// TIA Portal V19 export
FUNCTION_BLOCK "System_FB"   // FB3, LAD
TITLE = System bits
AUTHOR : Piemme
FAMILY : System
VERSION : 1.2
// stored: Access Published, MemoryReserve 100, SetENOAutomatically false
   VAR_INPUT
      PbLampTest : Bool;
   END_VAR
   VAR
      Ton0 : IEC_TIMER;
      wFrequencyGen : Word;
      wFrequencyLampTest : Word;
      PreviuosCycleTime : "CpuPreviuosCycleTime";
   END_VAR
   VAR_TEMP   // added for the SCL form of the ladder/FBD networks
      _w1 : Bool;
   END_VAR
BEGIN

REGION Network 1 (SCL): Info
   //=============================================================================
   //PM FORMING
   //-----------------------------------------------------------------------------
   // Library: StandardBlocks
   // Tested with: S7-1518TF
   // Engineering: TIA Portal V18
   // Restrictions: -
   // Requirements: S7-1500
   // Functionality: System management
   //
   // v1.0.0  28/12/2022 
   //=============================================================================
END_REGION

REGION Network 2: Set/Rst bits always true / false
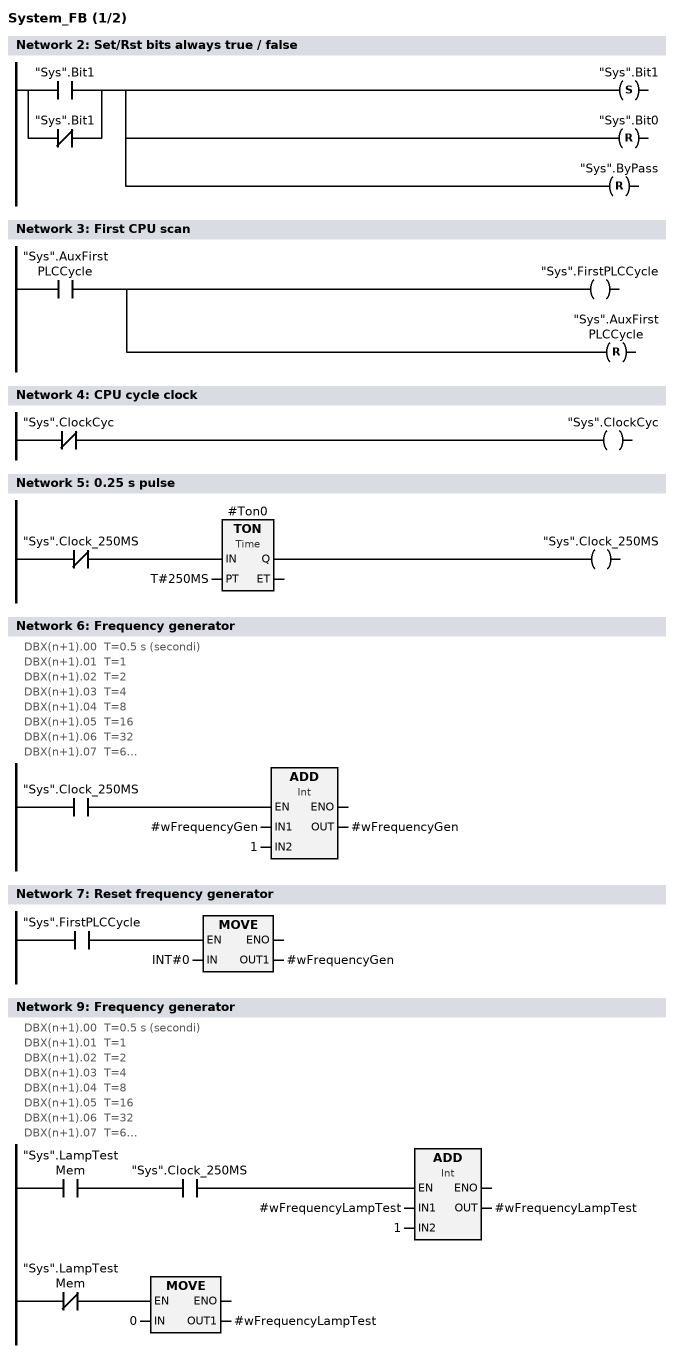
   RUNG wire#powerrail
      Contact( "Sys".Bit1 )
      wire#w1
      S_Coil( "Sys".Bit1 )
   END_RUNG
   RUNG wire#powerrail
      I_Contact( "Sys".Bit1 )
   END_RUNG wire#w1
   RUNG wire#w1
      R_Coil( "Sys".Bit0 )
   END_RUNG
   RUNG wire#w1
      R_Coil( "Sys".ByPass )
   END_RUNG
   // the same network as SCL:
   #_w1 := "Sys".Bit1 OR NOT "Sys".Bit1;
   IF #_w1 THEN
       "Sys".Bit1 := TRUE;
       "Sys".Bit0 := FALSE;
       "Sys".ByPass := FALSE;
   END_IF;
END_REGION

REGION Network 3: First CPU scan
   RUNG wire#powerrail
      Contact( "Sys".AuxFirstPLCCycle )
      wire#w1
      Coil( "Sys".FirstPLCCycle )
   END_RUNG
   RUNG wire#w1
      R_Coil( "Sys".AuxFirstPLCCycle )
   END_RUNG
   // the same network as SCL:
   "Sys".FirstPLCCycle := "Sys".AuxFirstPLCCycle;
   IF "Sys".AuxFirstPLCCycle THEN "Sys".AuxFirstPLCCycle := FALSE; END_IF;
END_REGION

REGION Network 4: CPU cycle clock
   RUNG wire#powerrail
      I_Contact( "Sys".ClockCyc )
      Coil( "Sys".ClockCyc )
   END_RUNG
   // the same network as SCL:
   "Sys".ClockCyc := NOT "Sys".ClockCyc;
END_REGION

REGION Network 5: 0.25 s pulse
   RUNG wire#powerrail
      I_Contact( "Sys".Clock_250MS )
      { S7_Templates := "time_type := Time" } #Ton0.TON(pt := T#250MS, et =>)
      Coil( "Sys".Clock_250MS )
   END_RUNG
   // the same network as SCL:
   #Ton0.TON(IN := NOT "Sys".Clock_250MS, PT := T#250MS);
   "Sys".Clock_250MS := #Ton0.Q;
END_REGION

REGION Network 6: Frequency generator
   // DBX(n+1).00  T=0.5 s (secondi)
   // DBX(n+1).01  T=1
   // DBX(n+1).02  T=2
   // DBX(n+1).03  T=4
   // DBX(n+1).04  T=8
   // DBX(n+1).05  T=16
   // DBX(n+1).06  T=32
   // DBX(n+1).07  T=64     
   // DBX  (n).00  T=128    (2 M)
   // DBX  (n).01  T=256    (4.2 M)
   // DBX  (n).02  T=512    (8.5 M)
   // DBX  (n).03  T=1024   (17 M)
   // DBX  (n).04  T=2048   (34.1 M)
   // DBX  (n).05  T=4096   (68.2 M)
   // DBX  (n).06  T=8192   (2 H)
   // DBX  (n).07  T=16384  (4 H)
   RUNG wire#powerrail
      Contact( "Sys".Clock_250MS )
      { S7_Templates := "SrcType := Int"; S7_GenerateENO := "TRUE" } Add(in1 := #wFrequencyGen, in2 := 1, out => #wFrequencyGen)
   END_RUNG
   // the same network as SCL:
   IF "Sys".Clock_250MS THEN #wFrequencyGen := #wFrequencyGen + 1; END_IF;
END_REGION

REGION Network 7: Reset frequency generator
   RUNG wire#powerrail
      Contact( "Sys".FirstPLCCycle )
      { S7_GenerateENO := "TRUE" } Move(in := INT#0, out1 => #wFrequencyGen)
   END_RUNG
   // the same network as SCL:
   IF "Sys".FirstPLCCycle THEN #wFrequencyGen := INT#0; END_IF;
END_REGION

REGION Network 8 (SCL): MB of clocks / Clocks
   "Sys".Clock_500MS := #wFrequencyGen.%X0;
   "Sys".Clock_1S := #wFrequencyGen.%X1;
   "Sys".Clock_2S := #wFrequencyGen.%X2;
   "Sys".Clock_4S := #wFrequencyGen.%X3;
   "Sys".Clock_8S := #wFrequencyGen.%X4;
   "Sys".Clock_16S := #wFrequencyGen.%X5;
   "Sys".Clock_32S := #wFrequencyGen.%X6;
   "Sys".Clock_64S := #wFrequencyGen.%X7;
END_REGION

REGION Network 9: Frequency generator
   // DBX(n+1).00  T=0.5 s (secondi)
   // DBX(n+1).01  T=1
   // DBX(n+1).02  T=2
   // DBX(n+1).03  T=4
   // DBX(n+1).04  T=8
   // DBX(n+1).05  T=16
   // DBX(n+1).06  T=32
   // DBX(n+1).07  T=64     
   // DBX  (n).00  T=128    (2 M)
   // DBX  (n).01  T=256    (4.2 M)
   // DBX  (n).02  T=512    (8.5 M)
   // DBX  (n).03  T=1024   (17 M)
   // DBX  (n).04  T=2048   (34.1 M)
   // DBX  (n).05  T=4096   (68.2 M)
   // DBX  (n).06  T=8192   (2 H)
   // DBX  (n).07  T=16384  (4 H)
   RUNG wire#powerrail
      Contact( "Sys".LampTestMem )
      Contact( "Sys".Clock_250MS )
      { S7_Templates := "SrcType := Int"; S7_GenerateENO := "TRUE" } Add(in1 := #wFrequencyLampTest, in2 := 1, out => #wFrequencyLampTest)
   END_RUNG
   RUNG wire#powerrail
      I_Contact( "Sys".LampTestMem )
      Move(in := 0, out1 => #wFrequencyLampTest)
   END_RUNG
   // the same network as SCL:
   IF "Sys".LampTestMem AND "Sys".Clock_250MS THEN #wFrequencyLampTest := #wFrequencyLampTest + 1; END_IF;
   IF NOT "Sys".LampTestMem THEN #wFrequencyLampTest := 0; END_IF;
END_REGION

REGION Network 10: Lamps Test
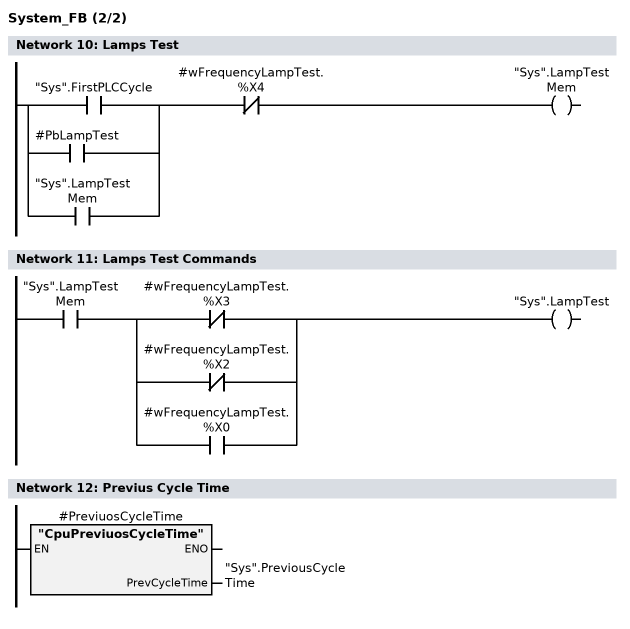
   RUNG wire#powerrail
      Contact( "Sys".FirstPLCCycle )
      wire#w1
      I_Contact( #wFrequencyLampTest.%X4 )
      Coil( "Sys".LampTestMem )
   END_RUNG
   RUNG wire#powerrail
      Contact( #PbLampTest )
   END_RUNG wire#w1
   RUNG wire#powerrail
      Contact( "Sys".LampTestMem )
   END_RUNG wire#w1
   // the same network as SCL:
   "Sys".LampTestMem := ("Sys".FirstPLCCycle OR #PbLampTest OR "Sys".LampTestMem) AND NOT #wFrequencyLampTest.%X4;
END_REGION

REGION Network 11: Lamps Test Commands
   RUNG wire#powerrail
      Contact( "Sys".LampTestMem )
      wire#w1
      I_Contact( #wFrequencyLampTest.%X3 )
      wire#w2
      Coil( "Sys".LampTest )
   END_RUNG
   RUNG wire#w1
      I_Contact( #wFrequencyLampTest.%X2 )
   END_RUNG wire#w2
   RUNG wire#w1
      Contact( #wFrequencyLampTest.%X0 )
   END_RUNG wire#w2
   // the same network as SCL:
   "Sys".LampTest := "Sys".LampTestMem AND (NOT #wFrequencyLampTest.%X3 OR NOT #wFrequencyLampTest.%X2 OR #wFrequencyLampTest.%X0);
END_REGION

REGION Network 12: Previus Cycle Time
   RUNG wire#powerrail
      #PreviuosCycleTime(PrevCycleTime => "Sys".PreviousCycleTime)
   END_RUNG
   // the same network as SCL:
   #PreviuosCycleTime(PrevCycleTime => "Sys".PreviousCycleTime);   // "CpuPreviuosCycleTime"
END_REGION
END_FUNCTION_BLOCK
